{attribute addProperty BoxType "EL6201-0000-0017"}
{attribute addProperty Id "Slave_30A_DO0BIT10.125233Slave_30A_DO1BIT10.125234Slave_30A_DO2BIT10.125235Slave_30A_DO3BIT10.125236Slave_30B_DO0BIT10.125237Slave_30B_DO1BIT10.125238Slave_30B_DO2BIT10.125239Slave_30B_DO3BIT10.125240"}
{attribute addProperty CRC "4234797935"}
{attribute addProperty SizeInBites "8"}
{attribute addProperty SizeInBytes "1"}
TYPE Slave_30_Outputs_FC69E36F :
STRUCT
	{attribute addProperty Name "Slave_30A_DO0"}
	Slave_30A_DO0 : BIT;
	{attribute addProperty Name "Slave_30A_DO1"}
	Slave_30A_DO1 : BIT;
	{attribute addProperty Name "Slave_30A_DO2"}
	Slave_30A_DO2 : BIT;
	{attribute addProperty Name "Slave_30A_DO3"}
	Slave_30A_DO3 : BIT;
	{attribute addProperty Name "Slave_30B_DO0"}
	Slave_30B_DO0 : BIT;
	{attribute addProperty Name "Slave_30B_DO1"}
	Slave_30B_DO1 : BIT;
	{attribute addProperty Name "Slave_30B_DO2"}
	Slave_30B_DO2 : BIT;
	{attribute addProperty Name "Slave_30B_DO3"}
	Slave_30B_DO3 : BIT;
END_STRUCT
END_TYPE

(* stored: Version 1.2.0.0, ProductVersion 3.1.4024.9
   DUT Slave_30_Outputs_FC69E36F: Id {a8c7db1e-dde9-44ae-a329-29290ed7ddf0} *)
